// TIA Portal project "Cuptor" (V15.1)

(* hardware
DEVICE "S71500/ET200MP station_1"  S7-1500 station
   slot 0: "Rail_0"  Rack  6ES7 590-1***0-0AA0
   slot 1: "PLC_1"  CPU 1513-1 PN  6ES7 513-1AL02-0AB0  V2.6
      slot 3: "CPU display_1"  6ES7591-1AA00-0AA0
DEVICE "HMI_1"  KTP900 Basic PN
   slot 0: "HMI_1"  KTP900 Basic PN  6AV2 123-2JB03-0AX0  15.1.0.0
   slot 1: "HMI_RT_1"  KTP900 Basic PN  6AV2 123-2JB03-0AX0  15.1.0.0
   slot 5: "HMI_1.IE_CP_1"  PROFINET Interface  15.0.1.0
      slot 1: "PROFINET Interface_1"  PROFINET Interface
         slot 1: "Port_1"  Port
*)

// ===== PLC "PLC_1"  CPU 1513-1 PN =====

VAR_GLOBAL   // PLC tag table "Default tag table"
   "Clock_Byte" AT %MB0 : Byte;
   "Clock_10Hz" AT %M0.0 : Bool;
   "Clock_5Hz" AT %M0.1 : Bool;
   "Clock_2.5Hz" AT %M0.2 : Bool;
   "Clock_2Hz" AT %M0.3 : Bool;
   "Clock_1.25Hz" AT %M0.4 : Bool;
   "Clock_1Hz" AT %M0.5 : Bool;
   "Clock_0.625Hz" AT %M0.6 : Bool;
   "Clock_0.5Hz" AT %M0.7 : Bool;
END_VAR

DATA_BLOCK "Avarii"   // DB1
{ S7_Optimized_Access := 'TRUE' }
VERSION : 0.1
   VAR
      esd : Bool;
      esd_btn : Bool;
      reset_esd_btn : Bool;
      avarie_usa : Bool;
      avarie_trapa : Bool;
      avarie_arzator : Bool;
      avarie_ventilator : Bool;
      avarie_generala : Bool;
      reset_avarie_generala_btn : Bool;
      avarie_hmi : Bool;
      "anti-viagra_pt_al7" : Bool;
   END_VAR
BEGIN
END_DATA_BLOCK

DATA_BLOCK "Usa"   // DB2
{ S7_Optimized_Access := 'TRUE' }
VERSION : 0.1
   VAR
      usa_inchisa : Bool;
      btn_usa_deschisa : Bool;
      btn_usa_deschidere_urgenta : Bool;
   END_VAR
BEGIN
END_DATA_BLOCK

DATA_BLOCK "Trapa"   // DB3
{ S7_Optimized_Access := 'TRUE' }
VERSION : 0.1
   VAR
      trapa_inchisa : Bool;
      btn_trapa_deschisa : Bool;
      btn_trapa_deschidere_urgenta : Bool;
   END_VAR
BEGIN
END_DATA_BLOCK

DATA_BLOCK "Arzator"   // DB4
{ S7_Optimized_Access := 'TRUE' }
VERSION : 0.1
   VAR
      btn_pornire : Bool;
      arzator_pornit : Bool;
   END_VAR
BEGIN
END_DATA_BLOCK

DATA_BLOCK "Ventilator"   // DB5
{ S7_Optimized_Access := 'TRUE' }
VERSION : 0.1
   VAR
      btn_pornire : Bool;
      btn_pornire_urgenta : Bool;
      pornire_stea : Bool;
      pornire_triunghi : Bool;
      pornire_ventilator : Bool;
   END_VAR
BEGIN
END_DATA_BLOCK

DATA_BLOCK "Alarme"   // DB6
{ S7_Optimized_Access := 'TRUE' }
VERSION : 0.1
   VAR
      alarm_gather : Word;
      alarm_vect : Array[0..15] of Bool;
   END_VAR
BEGIN
END_DATA_BLOCK

DATA_BLOCK "Permisiuni"   // DB7
{ S7_Optimized_Access := 'TRUE' }
VERSION : 0.1
   VAR
      permisiune_pornire : Bool;
      cuptor_terminat : Bool;
      timp_50 : Time;
      timp_80 : Time;
      auxiliar_alarma_7 : Bool;
   END_VAR
BEGIN
END_DATA_BLOCK

DATA_BLOCK "Simulare"   // DB10
{ S7_Optimized_Access := 'TRUE' }
VERSION : 0.1
   VAR
      temperatura_curenta : Real;
      temperatura_ceruta : Real;
      temperatura_deschidere : Real := 18.0;
      timp_cuptor : Time;
      resetare_cuptor : Bool;
      timp_curent : Time;
      timp_curent_hmi : Time;
      timp_cuptor_ms : Time;
      add_triunghi : Int;
      paritate_triunghi : Int;
      add_stea : Int;
      paritate_stea : Int;
   END_VAR
BEGIN
END_DATA_BLOCK

DATA_BLOCK "Butoane"   // DB11
{ S7_Optimized_Access := 'TRUE' }
VERSION : 0.1
   VAR
      btn_pornire : Bool;
      btn_pauza : Bool;
      btn_continuare : Bool;
      re_test : Bool;
   END_VAR
BEGIN
END_DATA_BLOCK

DATA_BLOCK "Usa_FB_DB"   // DB12
{ S7_Optimized_Access := 'TRUE' }
VERSION : 0.1
// stored: InstanceOfName Usa_FB
"Usa_FB"
BEGIN
END_DATA_BLOCK

DATA_BLOCK "Trapa_FB_DB"   // DB13
{ S7_Optimized_Access := 'TRUE' }
VERSION : 0.1
// stored: InstanceOfName Trapa_FB
"Trapa_FB"
BEGIN
END_DATA_BLOCK

DATA_BLOCK "Ventilator_FB_DB"   // DB14
{ S7_Optimized_Access := 'TRUE' }
VERSION : 0.1
// stored: InstanceOfName Ventilator_FB
"Ventilator_FB"
BEGIN
END_DATA_BLOCK

DATA_BLOCK "Arzator_FB_DB"   // DB16
{ S7_Optimized_Access := 'TRUE' }
VERSION : 0.1
// stored: InstanceOfName Arzator_FB
"Arzator_FB"
BEGIN
END_DATA_BLOCK

DATA_BLOCK "Simulare_FB_DB"   // DB17
{ S7_Optimized_Access := 'TRUE' }
VERSION : 0.1
// stored: InstanceOfName Simulare_FB
"Simulare_FB"
BEGIN
END_DATA_BLOCK

DATA_BLOCK "Hysteresis_DB_1"   // DB18
{ S7_Optimized_Access := 'TRUE' }
VERSION : 0.1
// stored: InstanceOfName Hysteresis
"Hysteresis"
BEGIN
END_DATA_BLOCK

DATA_BLOCK "Variabile_HMI"   // DB19
{ S7_Optimized_Access := 'TRUE' }
VERSION : 0.1
   VAR
      re_stea : Bool;
      re_triunghi : Bool;
      stea_1 : Bool;
      triunghi_1 : Bool;
      triunghi_2 : Bool;
      stea_2 : Bool;
   END_VAR
BEGIN
END_DATA_BLOCK

// folder: System blocks/Program resources

DATA_BLOCK "Reset_esd"   // DB8
{ S7_Optimized_Access := 'TRUE' }
AUTHOR : Simatic
FAMILY : IEC
NAME : IEC_TMR
VERSION : 1.0
// stored: InstanceOfName IEC_TIMER
"IEC_TIMER"
BEGIN
END_DATA_BLOCK

DATA_BLOCK "Reset_avarie_generala"   // DB9
{ S7_Optimized_Access := 'TRUE' }
AUTHOR : Simatic
FAMILY : IEC
NAME : IEC_TMR
VERSION : 1.0
// stored: InstanceOfName IEC_TIMER
"IEC_TIMER"
BEGIN
END_DATA_BLOCK

DATA_BLOCK "restart_btn_pornire"   // DB15
{ S7_Optimized_Access := 'TRUE' }
AUTHOR : Simatic
FAMILY : IEC
NAME : IEC_TMR
VERSION : 1.0
// stored: InstanceOfName IEC_TIMER
"IEC_TIMER"
BEGIN
END_DATA_BLOCK

// folder: (top level)

FUNCTION_BLOCK "Usa_FB"   // FB1, LAD
{ S7_Optimized_Access := 'TRUE' }
VERSION : 0.1
   VAR_INPUT
      esd : Bool;
      avarie : Bool;
      btn_deschidere_urgenta : Bool;
      temperatura_curenta : Real;
      temperatura_deschidere : Real;
   END_VAR
   VAR_OUTPUT
      usa_inchisa : Bool;
      alarma : Bool;
   END_VAR
   VAR_IN_OUT
      btn_deschidere : Bool;
   END_VAR
   VAR
      timer_reset_alarma : TON_TIME;
   END_VAR
BEGIN

REGION Network 1: Deschide usa(normal sau extrem)
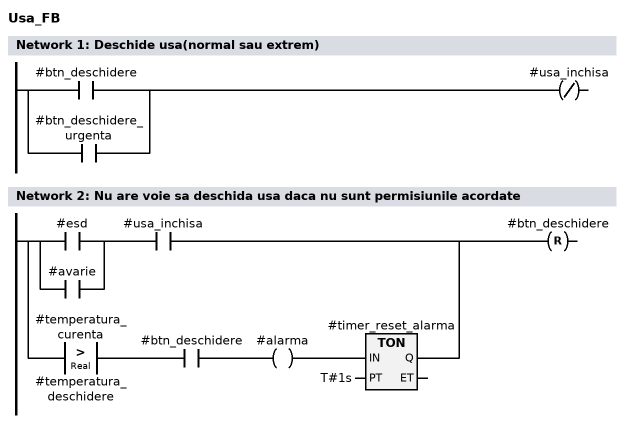
   RUNG wire#powerrail
      Contact( #btn_deschidere )
      wire#w1
      I_Coil( #usa_inchisa )
   END_RUNG
   RUNG wire#powerrail
      Contact( #btn_deschidere_urgenta )
   END_RUNG wire#w1
   // the same network as SCL:
   #usa_inchisa := NOT (#btn_deschidere OR #btn_deschidere_urgenta);
END_REGION

REGION Network 2: Nu are voie sa deschida usa daca nu sunt permisiunile acordate
   #alarma := (#temperatura_curenta > #temperatura_deschidere) AND #btn_deschidere;
   #timer_reset_alarma(IN := #alarma, PT := T#1s);   // TON
   IF ((#esd OR #avarie) AND #usa_inchisa) OR #timer_reset_alarma.Q THEN #btn_deschidere := FALSE; END_IF;
END_REGION
END_FUNCTION_BLOCK

FUNCTION_BLOCK "Trapa_FB"   // FB2, LAD
{ S7_Optimized_Access := 'TRUE' }
VERSION : 0.1
   VAR_INPUT
      esd : Bool;
      avarie : Bool;
      btn_deschidere_urgenta : Bool;
      cuptor_terminat : Bool;
      temperatura_curenta : Real;
      temperatura_inchidere_trapa : Real;
   END_VAR
   VAR_OUTPUT
      trapa_inchisa : Bool;
   END_VAR
   VAR_IN_OUT
      btn_deschidere : Bool;
   END_VAR
BEGIN

REGION Network 1: Deschide trapa(normla si urgenta)
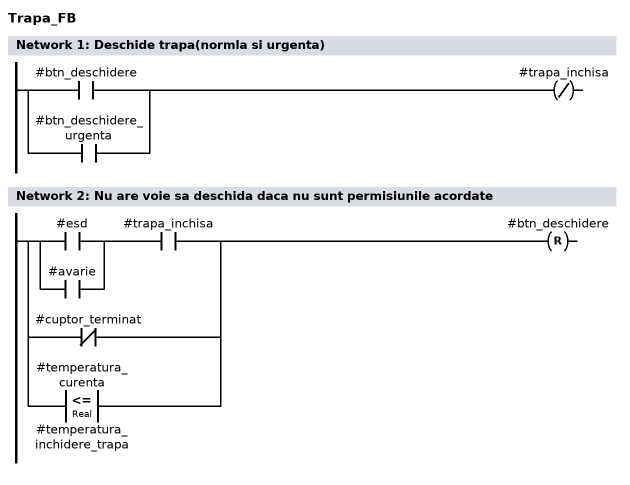
   RUNG wire#powerrail
      Contact( #btn_deschidere )
      wire#w1
      I_Coil( #trapa_inchisa )
   END_RUNG
   RUNG wire#powerrail
      Contact( #btn_deschidere_urgenta )
   END_RUNG wire#w1
   // the same network as SCL:
   #trapa_inchisa := NOT (#btn_deschidere OR #btn_deschidere_urgenta);
END_REGION

REGION Network 2: Nu are voie sa deschida daca nu sunt permisiunile acordate
   RUNG wire#powerrail
      Contact( #esd )
      wire#w1
      Contact( #trapa_inchisa )
      wire#w2
      R_Coil( #btn_deschidere )
   END_RUNG
   RUNG wire#powerrail
      Contact( #avarie )
   END_RUNG wire#w1
   RUNG wire#powerrail
      I_Contact( #cuptor_terminat )
   END_RUNG wire#w2
   RUNG wire#powerrail
      { S7_Templates := "SrcType := Real" } LE_Contact(in1 := #temperatura_curenta, in2 := #temperatura_inchidere_trapa)
   END_RUNG wire#w2
   // the same network as SCL:
   IF ((#esd OR #avarie) AND #trapa_inchisa) OR NOT #cuptor_terminat OR (#temperatura_curenta <= #temperatura_inchidere_trapa) THEN
       #btn_deschidere := FALSE;
   END_IF;
END_REGION
END_FUNCTION_BLOCK

FUNCTION_BLOCK "Arzator_FB"   // FB3, LAD
{ S7_Optimized_Access := 'TRUE' }
VERSION : 0.1
   VAR_INPUT
      esd : Bool;
      avarie : Bool;
      temperatura_curenta : Real;
      temperatura_dorita : Real;
   END_VAR
   VAR_OUTPUT
      pornire_arzator : Bool;
   END_VAR
   VAR_IN_OUT
      btn_pornire : Bool;
   END_VAR
BEGIN

REGION Network 1: Porneste valva
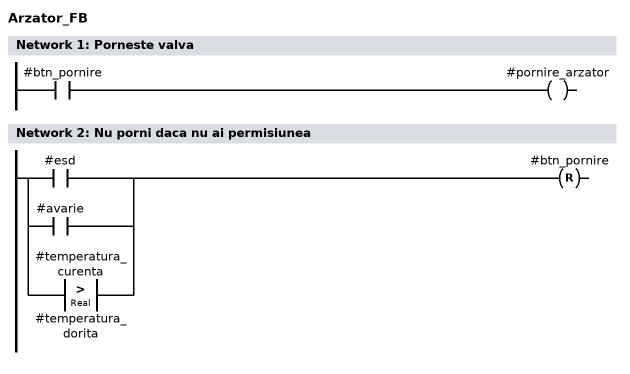
   RUNG wire#powerrail
      Contact( #btn_pornire )
      Coil( #pornire_arzator )
   END_RUNG
   // the same network as SCL:
   #pornire_arzator := #btn_pornire;
END_REGION

REGION Network 2: Nu porni daca nu ai permisiunea
   RUNG wire#powerrail
      Contact( #esd )
      wire#w1
      R_Coil( #btn_pornire )
   END_RUNG
   RUNG wire#powerrail
      Contact( #avarie )
   END_RUNG wire#w1
   RUNG wire#powerrail
      { S7_Templates := "SrcType := Real" } GT_Contact(in1 := #temperatura_curenta, in2 := #temperatura_dorita)
   END_RUNG wire#w1
   // the same network as SCL:
   IF #esd OR #avarie OR (#temperatura_curenta > #temperatura_dorita) THEN #btn_pornire := FALSE; END_IF;
END_REGION
END_FUNCTION_BLOCK

FUNCTION_BLOCK "Ventilator_FB"   // FB4, LAD
{ S7_Optimized_Access := 'TRUE' }
VERSION : 0.1
   VAR_INPUT
      esd : Bool;
      avarie : Bool;
      cuptor_terminat : Bool;
      btn_pornire_urgenta : Bool;
      temperatura_curenta : Real;
      temperatura_inchidere_ventilator : Real;
   END_VAR
   VAR_OUTPUT
      pornire_ventilator_stea : Bool;
      pornire_ventilator_triunghi : Bool;
      ventilator_pornit : Bool;
   END_VAR
   VAR_IN_OUT
      btn_pornire : Bool;
   END_VAR
   VAR
      timer_stea : TON_TIME;
   END_VAR
BEGIN

REGION Network 1: Porneste ventilatorul(normal si urgenta)
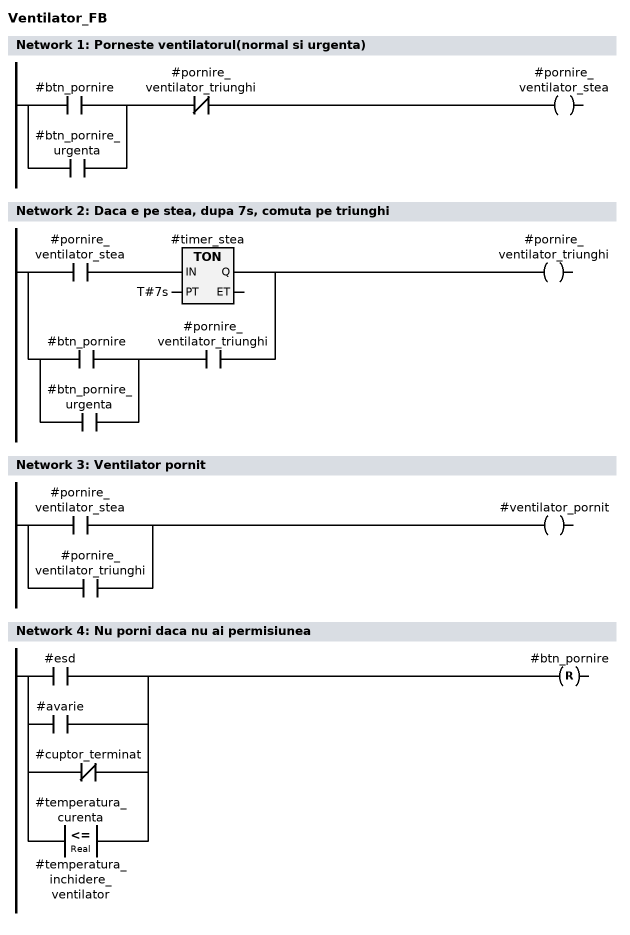
   RUNG wire#powerrail
      Contact( #btn_pornire )
      wire#w1
      I_Contact( #pornire_ventilator_triunghi )
      Coil( #pornire_ventilator_stea )
   END_RUNG
   RUNG wire#powerrail
      Contact( #btn_pornire_urgenta )
   END_RUNG wire#w1
   // the same network as SCL:
   #pornire_ventilator_stea := (#btn_pornire OR #btn_pornire_urgenta) AND NOT #pornire_ventilator_triunghi;
END_REGION

REGION Network 2: Daca e pe stea, dupa 7s, comuta pe triunghi
   #timer_stea(IN := #pornire_ventilator_stea, PT := T#7s);   // TON
   #pornire_ventilator_triunghi := #timer_stea.Q OR ((#btn_pornire OR #btn_pornire_urgenta) AND #pornire_ventilator_triunghi);
END_REGION

REGION Network 3: Ventilator pornit
   RUNG wire#powerrail
      Contact( #pornire_ventilator_stea )
      wire#w1
      Coil( #ventilator_pornit )
   END_RUNG
   RUNG wire#powerrail
      Contact( #pornire_ventilator_triunghi )
   END_RUNG wire#w1
   // the same network as SCL:
   #ventilator_pornit := #pornire_ventilator_stea OR #pornire_ventilator_triunghi;
END_REGION

REGION Network 4: Nu porni daca nu ai permisiunea
   RUNG wire#powerrail
      Contact( #esd )
      wire#w1
      R_Coil( #btn_pornire )
   END_RUNG
   RUNG wire#powerrail
      Contact( #avarie )
   END_RUNG wire#w1
   RUNG wire#powerrail
      I_Contact( #cuptor_terminat )
   END_RUNG wire#w1
   RUNG wire#powerrail
      { S7_Templates := "SrcType := Real" } LE_Contact(in1 := #temperatura_curenta, in2 := #temperatura_inchidere_ventilator)
   END_RUNG wire#w1
   // the same network as SCL:
   IF #esd OR #avarie OR NOT #cuptor_terminat OR (#temperatura_curenta <= #temperatura_inchidere_ventilator) THEN
       #btn_pornire := FALSE;
   END_IF;
END_REGION
END_FUNCTION_BLOCK

FUNCTION_BLOCK "Simulare_FB"   // FB5, LAD
{ S7_Optimized_Access := 'TRUE' }
VERSION : 0.1
   VAR_INPUT
      esd : Bool;
      avarie : Bool;
      temp_dorita : Real;
      temp_mediu : Real := 0.0;
      timp_cuptor : Time;
      trapa : Bool;
      ventilator : Bool;
      ventilator_stea : Bool;
      ventilator_triunghi : Bool;
   END_VAR
   VAR_OUTPUT
      timp_curent : Time;
      btn_trapa : Bool;
      btn_ventilator : Bool;
      terminat : Bool;
      alarma : Bool;
   END_VAR
   VAR_IN_OUT
      resetare_cuptor : Bool;
      temp_curenta : Real;
      pornire_arzator : Bool;
      conditie_pornire : Bool;
   END_VAR
   VAR
      timp_curent_secunde : Time;
      timer_cuptor : TON_TIME;
      re1 : Bool;
      re2 : Bool;
      timp_terminat : Bool;
      temp_in_limite : Bool;
      timer_reset_btn_resetare_cuptor : TON_TIME;
   END_VAR
   VAR_TEMP   // added for the SCL form of the ladder/FBD networks
      _w1 : Bool;
      _w2 : Bool;
      _w3 : Bool;
   END_VAR
BEGIN

REGION Network 1: Daca are permisiunea, da drumul la valva
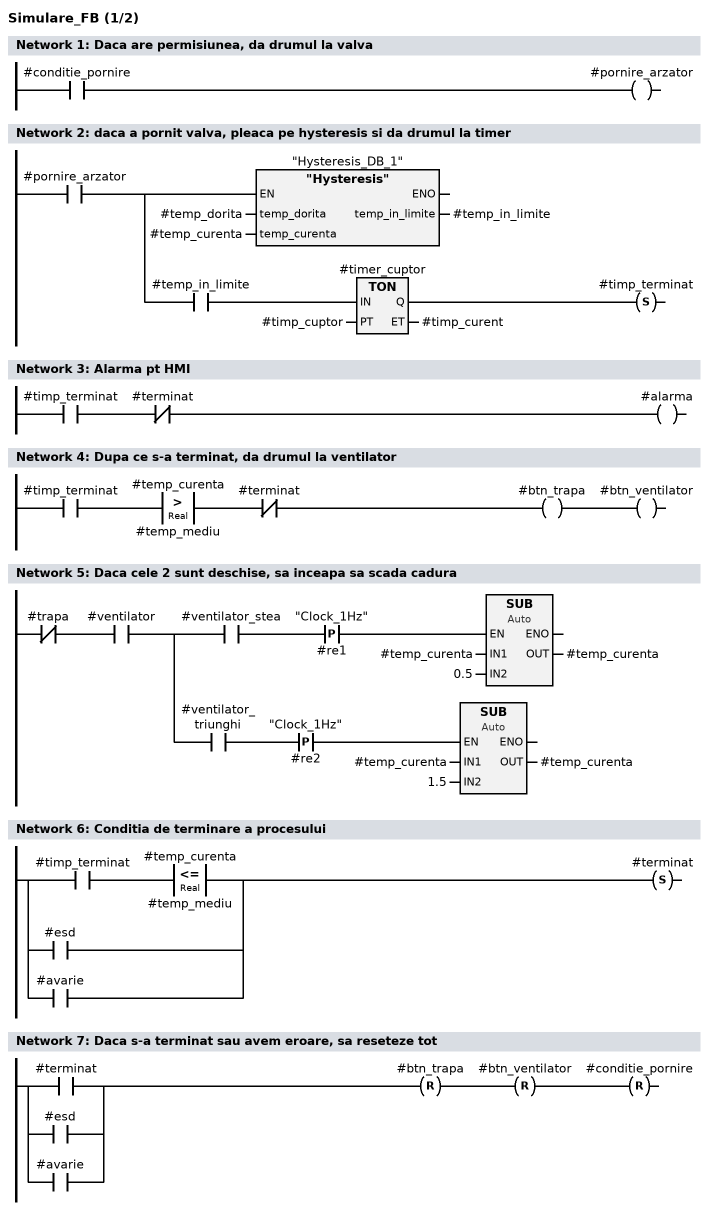
   RUNG wire#powerrail
      Contact( #conditie_pornire )
      Coil( #pornire_arzator )
   END_RUNG
   // the same network as SCL:
   #pornire_arzator := #conditie_pornire;
END_REGION

REGION Network 2: daca a pornit valva, pleaca pe hysteresis si da drumul la timer
   IF #pornire_arzator THEN
       "Hysteresis_DB_1"(temp_dorita := #temp_dorita,   // "Hysteresis"
                         temp_curenta := #temp_curenta,
                         temp_in_limite => #temp_in_limite);
   END_IF;
   #timer_cuptor(IN := #pornire_arzator AND #temp_in_limite, PT := #timp_cuptor, ET => #timp_curent);   // TON
   IF #timer_cuptor.Q THEN #timp_terminat := TRUE; END_IF;
END_REGION

REGION Network 3: Alarma pt HMI
   RUNG wire#powerrail
      Contact( #timp_terminat )
      I_Contact( #terminat )
      Coil( #alarma )
   END_RUNG
   // the same network as SCL:
   #alarma := #timp_terminat AND NOT #terminat;
END_REGION

REGION Network 4: Dupa ce s-a terminat, da drumul la ventilator
   RUNG wire#powerrail
      Contact( #timp_terminat )
      { S7_Templates := "SrcType := Real" } GT_Contact(in1 := #temp_curenta, in2 := #temp_mediu)
      I_Contact( #terminat )
      Coil( #btn_trapa )
      Coil( #btn_ventilator )
   END_RUNG
   // the same network as SCL:
   #btn_trapa := #timp_terminat AND (#temp_curenta > #temp_mediu) AND NOT #terminat;
   #btn_ventilator := #btn_trapa;
END_REGION

REGION Network 5: Daca cele 2 sunt deschise, sa inceapa sa scada cadura
   RUNG wire#powerrail
      I_Contact( #trapa )
      Contact( #ventilator )
      wire#w1
      Contact( #ventilator_stea )
      P_Contact(operand := "Clock_1Hz", bit := #re1)
      Sub(in1 := #temp_curenta, in2 := 0.5, out => #temp_curenta)
   END_RUNG
   RUNG wire#w1
      Contact( #ventilator_triunghi )
      P_Contact(operand := "Clock_1Hz", bit := #re2)
      Sub(in1 := #temp_curenta, in2 := 1.5, out => #temp_curenta)
   END_RUNG
   // the same network as SCL:
   #_w1 := NOT #trapa AND #ventilator;
   #_w2 := #_w1 AND #ventilator_stea AND "Clock_1Hz" AND NOT #re1;   // rising edge of "Clock_1Hz"
   #re1 := "Clock_1Hz";
   IF #_w2 THEN #temp_curenta := #temp_curenta - 0.5; END_IF;
   #_w3 := #_w1 AND #ventilator_triunghi AND "Clock_1Hz" AND NOT #re2;   // rising edge of "Clock_1Hz"
   #re2 := "Clock_1Hz";
   IF #_w3 THEN #temp_curenta := #temp_curenta - 1.5; END_IF;
END_REGION

REGION Network 6: Conditia de terminare a procesului
   RUNG wire#powerrail
      Contact( #timp_terminat )
      { S7_Templates := "SrcType := Real" } LE_Contact(in1 := #temp_curenta, in2 := #temp_mediu)
      wire#w1
      S_Coil( #terminat )
   END_RUNG
   RUNG wire#powerrail
      Contact( #esd )
   END_RUNG wire#w1
   RUNG wire#powerrail
      Contact( #avarie )
   END_RUNG wire#w1
   // the same network as SCL:
   IF (#timp_terminat AND (#temp_curenta <= #temp_mediu)) OR #esd OR #avarie THEN #terminat := TRUE; END_IF;
END_REGION

REGION Network 7: Daca s-a terminat sau avem eroare, sa reseteze tot
   RUNG wire#powerrail
      Contact( #terminat )
      wire#w1
      R_Coil( #btn_trapa )
      R_Coil( #btn_ventilator )
      R_Coil( #conditie_pornire )
   END_RUNG
   RUNG wire#powerrail
      Contact( #esd )
   END_RUNG wire#w1
   RUNG wire#powerrail
      Contact( #avarie )
   END_RUNG wire#w1
   // the same network as SCL:
   IF #terminat OR #esd OR #avarie THEN
       #btn_trapa := FALSE;
       #btn_ventilator := FALSE;
       #conditie_pornire := FALSE;
   END_IF;
END_REGION

REGION Network 8: Resetare cuptor
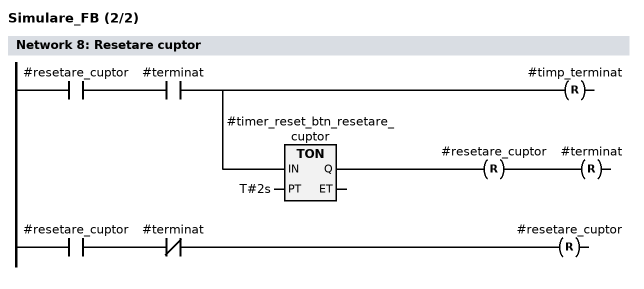
   #_w1 := #resetare_cuptor AND #terminat;
   IF #_w1 THEN #timp_terminat := FALSE; END_IF;
   #timer_reset_btn_resetare_cuptor(IN := #_w1, PT := T#2s);   // TON
   IF #timer_reset_btn_resetare_cuptor.Q THEN
       #resetare_cuptor := FALSE;
       #terminat := FALSE;
   END_IF;
   IF #resetare_cuptor AND NOT #terminat THEN #resetare_cuptor := FALSE; END_IF;
END_REGION
END_FUNCTION_BLOCK

FUNCTION_BLOCK "Hysteresis"   // FB6, LAD
{ S7_Optimized_Access := 'TRUE' }
VERSION : 0.1
   VAR_INPUT
      temp_dorita : Real;
   END_VAR
   VAR_OUTPUT
      temp_in_limite : Bool;
   END_VAR
   VAR_IN_OUT
      temp_curenta : Real;
   END_VAR
   VAR
      crestere_temp : Real := 0.5;
      limita_inferioara : Real;
      limita_superioara : Real;
      differenta_pt_limite : Real := 2.0;
      re1 : Bool;
      re2 : Bool;
      urcare : Bool;
      coborare : Bool;
   END_VAR
   VAR_TEMP   // added for the SCL form of the ladder/FBD networks
      _w1 : Bool;
   END_VAR
BEGIN

REGION Network 1: Calcul pentru limite
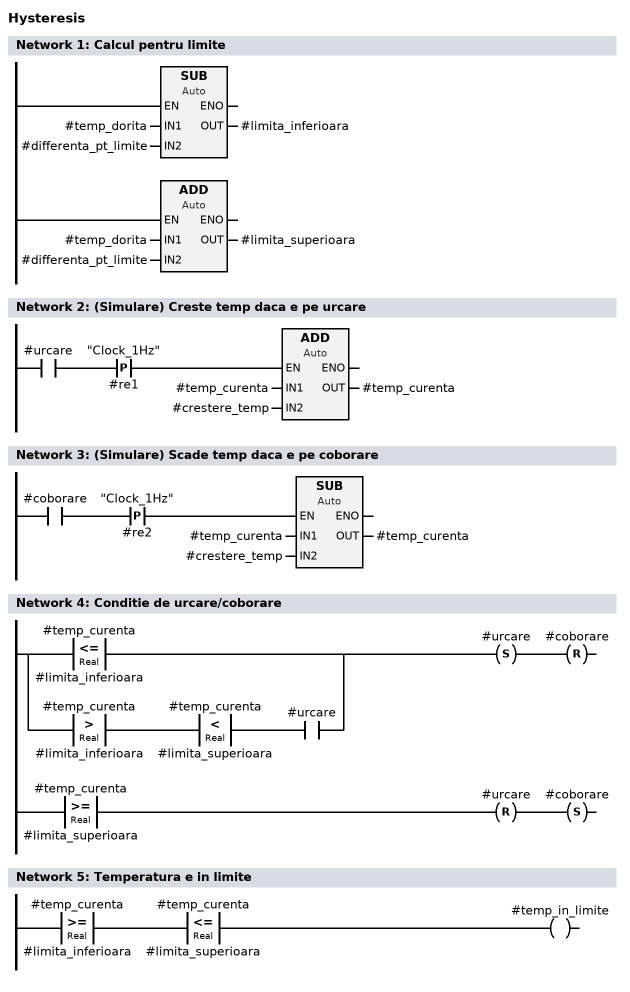
   RUNG wire#powerrail
      Sub(in1 := #temp_dorita, in2 := #differenta_pt_limite, out => #limita_inferioara)
   END_RUNG
   RUNG wire#powerrail
      Add(in1 := #temp_dorita, in2 := #differenta_pt_limite, out => #limita_superioara)
   END_RUNG
   // the same network as SCL:
   #limita_inferioara := #temp_dorita - #differenta_pt_limite;
   #limita_superioara := #temp_dorita + #differenta_pt_limite;
END_REGION

REGION Network 2: (Simulare) Creste temp daca e pe urcare
   RUNG wire#powerrail
      Contact( #urcare )
      P_Contact(operand := "Clock_1Hz", bit := #re1)
      Add(in1 := #temp_curenta, in2 := #crestere_temp, out => #temp_curenta)
   END_RUNG
   // the same network as SCL:
   #_w1 := #urcare AND "Clock_1Hz" AND NOT #re1;   // rising edge of "Clock_1Hz"
   #re1 := "Clock_1Hz";
   IF #_w1 THEN #temp_curenta := #temp_curenta + #crestere_temp; END_IF;
END_REGION

REGION Network 3: (Simulare) Scade temp daca e pe coborare
   RUNG wire#powerrail
      Contact( #coborare )
      P_Contact(operand := "Clock_1Hz", bit := #re2)
      Sub(in1 := #temp_curenta, in2 := #crestere_temp, out => #temp_curenta)
   END_RUNG
   // the same network as SCL:
   #_w1 := #coborare AND "Clock_1Hz" AND NOT #re2;   // rising edge of "Clock_1Hz"
   #re2 := "Clock_1Hz";
   IF #_w1 THEN #temp_curenta := #temp_curenta - #crestere_temp; END_IF;
END_REGION

REGION Network 4: Conditie de urcare/coborare
   RUNG wire#powerrail
      { S7_Templates := "SrcType := Real" } LE_Contact(in1 := #temp_curenta, in2 := #limita_inferioara)
      wire#w1
      S_Coil( #urcare )
      R_Coil( #coborare )
   END_RUNG
   RUNG wire#powerrail
      { S7_Templates := "SrcType := Real" } GT_Contact(in1 := #temp_curenta, in2 := #limita_inferioara)
      { S7_Templates := "SrcType := Real" } LT_Contact(in1 := #temp_curenta, in2 := #limita_superioara)
      Contact( #urcare )
   END_RUNG wire#w1
   RUNG wire#powerrail
      { S7_Templates := "SrcType := Real" } GE_Contact(in1 := #temp_curenta, in2 := #limita_superioara)
      R_Coil( #urcare )
      S_Coil( #coborare )
   END_RUNG
   // the same network as SCL:
   #_w1 := (#temp_curenta <= #limita_inferioara) OR ((#temp_curenta > #limita_inferioara) AND (#temp_curenta < #limita_superioara) AND #urcare);
   IF #_w1 THEN
       #urcare := TRUE;
       #coborare := FALSE;
   END_IF;
   IF #temp_curenta >= #limita_superioara THEN
       #urcare := FALSE;
       #coborare := TRUE;
   END_IF;
END_REGION

REGION Network 5: Temperatura e in limite
   RUNG wire#powerrail
      { S7_Templates := "SrcType := Real" } GE_Contact(in1 := #temp_curenta, in2 := #limita_inferioara)
      { S7_Templates := "SrcType := Real" } LE_Contact(in1 := #temp_curenta, in2 := #limita_superioara)
      Coil( #temp_in_limite )
   END_RUNG
   // the same network as SCL:
   #temp_in_limite := (#temp_curenta >= #limita_inferioara) AND (#temp_curenta <= #limita_superioara);
END_REGION
END_FUNCTION_BLOCK

ORGANIZATION_BLOCK "Main"   // OB1, LAD, ProgramCycle
TITLE = "Main Program Sweep (Cycle)"
{ S7_Optimized_Access := 'TRUE' }
VERSION : 0.1
   VAR_INPUT
      Initial_Call : Bool;   // Initial call of this OB
      Remanence : Bool;   // =True, if remanent data are available
   END_VAR
   VAR_TEMP   // added for the SCL form of the ladder/FBD networks
      _w1 : Bool;
      _w2 : Bool;
   END_VAR
BEGIN

REGION Network 1: Gather pt alarme
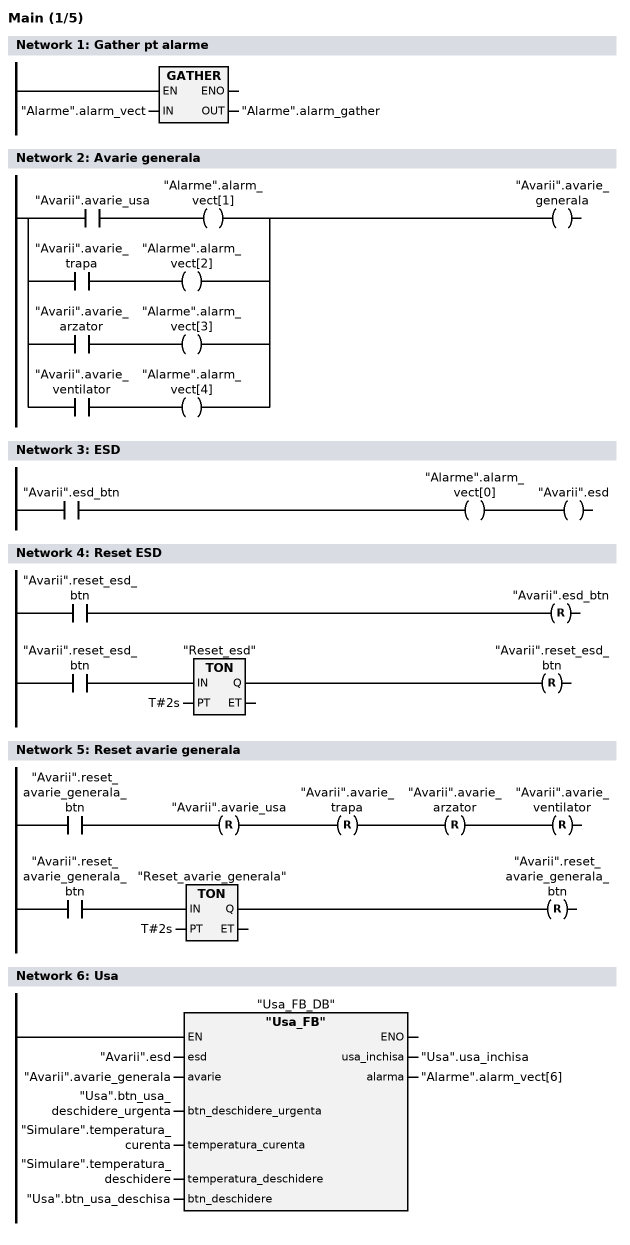
   GATHER(IN := "Alarme".alarm_vect, OUT => "Alarme".alarm_gather);
END_REGION

REGION Network 2: Avarie generala
   RUNG wire#powerrail
      Contact( "Avarii".avarie_usa )
      Coil( "Alarme".alarm_vect[1] )
      wire#w1
      Coil( "Avarii".avarie_generala )
   END_RUNG
   RUNG wire#powerrail
      Contact( "Avarii".avarie_trapa )
      Coil( "Alarme".alarm_vect[2] )
   END_RUNG wire#w1
   RUNG wire#powerrail
      Contact( "Avarii".avarie_arzator )
      Coil( "Alarme".alarm_vect[3] )
   END_RUNG wire#w1
   RUNG wire#powerrail
      Contact( "Avarii".avarie_ventilator )
      Coil( "Alarme".alarm_vect[4] )
   END_RUNG wire#w1
   // the same network as SCL:
   "Alarme".alarm_vect[1] := "Avarii".avarie_usa;
   "Alarme".alarm_vect[2] := "Avarii".avarie_trapa;
   "Alarme".alarm_vect[3] := "Avarii".avarie_arzator;
   "Alarme".alarm_vect[4] := "Avarii".avarie_ventilator;
   "Avarii".avarie_generala := "Avarii".avarie_usa OR "Avarii".avarie_trapa OR "Avarii".avarie_arzator OR "Avarii".avarie_ventilator;
END_REGION

REGION Network 3: ESD
   RUNG wire#powerrail
      Contact( "Avarii".esd_btn )
      Coil( "Alarme".alarm_vect[0] )
      Coil( "Avarii".esd )
   END_RUNG
   // the same network as SCL:
   "Alarme".alarm_vect[0] := "Avarii".esd_btn;
   "Avarii".esd := "Avarii".esd_btn;
END_REGION

REGION Network 4: Reset ESD
   IF "Avarii".reset_esd_btn THEN "Avarii".esd_btn := FALSE; END_IF;
   "Reset_esd".TON(IN := "Avarii".reset_esd_btn, PT := T#2s);
   IF "Reset_esd".Q THEN "Avarii".reset_esd_btn := FALSE; END_IF;
END_REGION

REGION Network 5: Reset avarie generala
   IF "Avarii".reset_avarie_generala_btn THEN
       "Avarii".avarie_usa := FALSE;
       "Avarii".avarie_trapa := FALSE;
       "Avarii".avarie_arzator := FALSE;
       "Avarii".avarie_ventilator := FALSE;
   END_IF;
   "Reset_avarie_generala".TON(IN := "Avarii".reset_avarie_generala_btn, PT := T#2s);
   IF "Reset_avarie_generala".Q THEN "Avarii".reset_avarie_generala_btn := FALSE; END_IF;
END_REGION

REGION Network 6: Usa
   RUNG wire#powerrail
      "Usa_FB_DB"(esd := "Avarii".esd, avarie := "Avarii".avarie_generala, btn_deschidere_urgenta := "Usa".btn_usa_deschidere_urgenta, temperatura_curenta := "Simulare".temperatura_curenta, temperatura_deschidere := "Simulare".temperatura_deschidere, btn_deschidere := "Usa".btn_usa_deschisa, usa_inchisa => "Usa".usa_inchisa, alarma => "Alarme".alarm_vect[6])
   END_RUNG
   // the same network as SCL:
   "Usa_FB_DB"(esd := "Avarii".esd,   // "Usa_FB"
               avarie := "Avarii".avarie_generala,
               btn_deschidere_urgenta := "Usa".btn_usa_deschidere_urgenta,
               temperatura_curenta := "Simulare".temperatura_curenta,
               temperatura_deschidere := "Simulare".temperatura_deschidere,
               btn_deschidere := "Usa".btn_usa_deschisa,
               usa_inchisa => "Usa".usa_inchisa,
               alarma => "Alarme".alarm_vect[6]);
END_REGION

REGION Network 7: Trapa
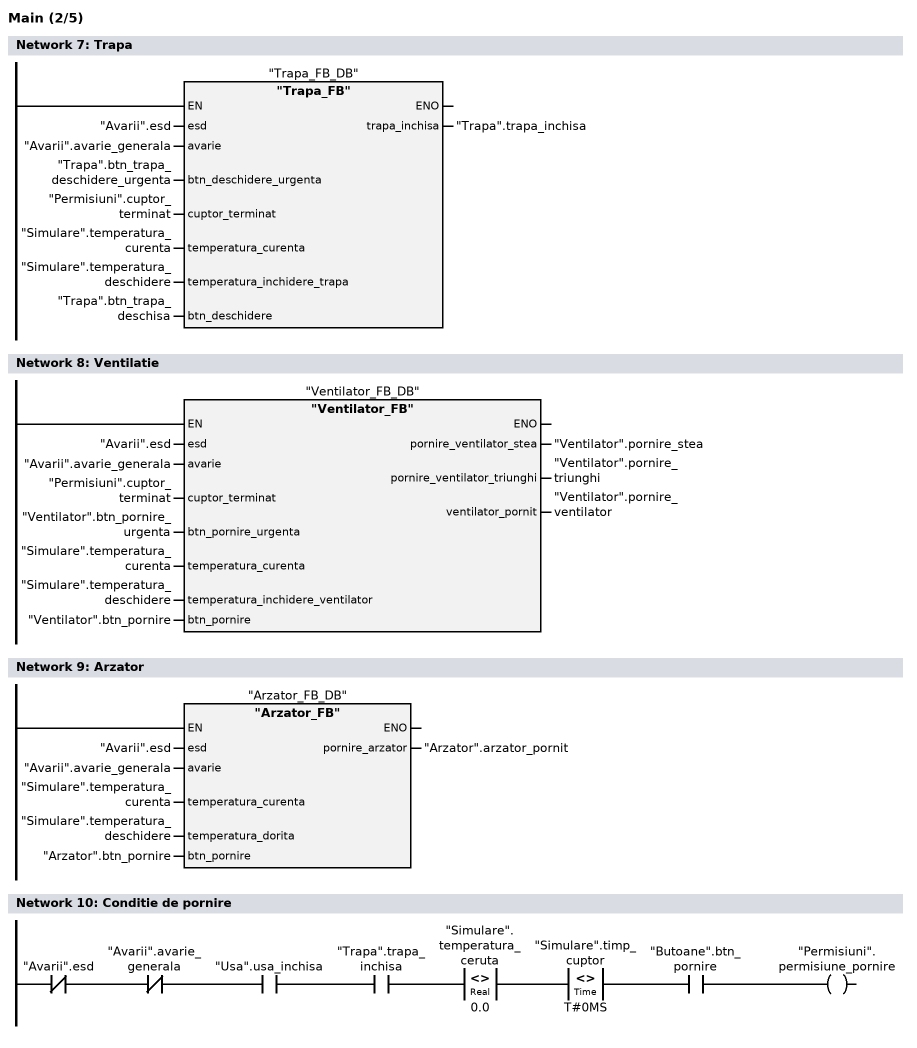
   RUNG wire#powerrail
      "Trapa_FB_DB"(esd := "Avarii".esd, avarie := "Avarii".avarie_generala, btn_deschidere_urgenta := "Trapa".btn_trapa_deschidere_urgenta, cuptor_terminat := "Permisiuni".cuptor_terminat, temperatura_curenta := "Simulare".temperatura_curenta, temperatura_inchidere_trapa := "Simulare".temperatura_deschidere, btn_deschidere := "Trapa".btn_trapa_deschisa, trapa_inchisa => "Trapa".trapa_inchisa)
   END_RUNG
   // the same network as SCL:
   "Trapa_FB_DB"(esd := "Avarii".esd,   // "Trapa_FB"
                 avarie := "Avarii".avarie_generala,
                 btn_deschidere_urgenta := "Trapa".btn_trapa_deschidere_urgenta,
                 cuptor_terminat := "Permisiuni".cuptor_terminat,
                 temperatura_curenta := "Simulare".temperatura_curenta,
                 temperatura_inchidere_trapa := "Simulare".temperatura_deschidere,
                 btn_deschidere := "Trapa".btn_trapa_deschisa,
                 trapa_inchisa => "Trapa".trapa_inchisa);
END_REGION

REGION Network 8: Ventilatie
   RUNG wire#powerrail
      "Ventilator_FB_DB"(esd := "Avarii".esd, avarie := "Avarii".avarie_generala, cuptor_terminat := "Permisiuni".cuptor_terminat, btn_pornire_urgenta := "Ventilator".btn_pornire_urgenta, temperatura_curenta := "Simulare".temperatura_curenta, temperatura_inchidere_ventilator := "Simulare".temperatura_deschidere, btn_pornire := "Ventilator".btn_pornire, pornire_ventilator_stea => "Ventilator".pornire_stea, pornire_ventilator_triunghi => "Ventilator".pornire_triunghi, ventilator_pornit => "Ventilator".pornire_ventilator)
   END_RUNG
   // the same network as SCL:
   "Ventilator_FB_DB"(esd := "Avarii".esd,   // "Ventilator_FB"
                      avarie := "Avarii".avarie_generala,
                      cuptor_terminat := "Permisiuni".cuptor_terminat,
                      btn_pornire_urgenta := "Ventilator".btn_pornire_urgenta,
                      temperatura_curenta := "Simulare".temperatura_curenta,
                      temperatura_inchidere_ventilator := "Simulare".temperatura_deschidere,
                      btn_pornire := "Ventilator".btn_pornire,
                      pornire_ventilator_stea => "Ventilator".pornire_stea,
                      pornire_ventilator_triunghi => "Ventilator".pornire_triunghi,
                      ventilator_pornit => "Ventilator".pornire_ventilator);
END_REGION

REGION Network 9: Arzator
   RUNG wire#powerrail
      "Arzator_FB_DB"(esd := "Avarii".esd, avarie := "Avarii".avarie_generala, temperatura_curenta := "Simulare".temperatura_curenta, temperatura_dorita := "Simulare".temperatura_deschidere, btn_pornire := "Arzator".btn_pornire, pornire_arzator => "Arzator".arzator_pornit)
   END_RUNG
   // the same network as SCL:
   "Arzator_FB_DB"(esd := "Avarii".esd,   // "Arzator_FB"
                   avarie := "Avarii".avarie_generala,
                   temperatura_curenta := "Simulare".temperatura_curenta,
                   temperatura_dorita := "Simulare".temperatura_deschidere,
                   btn_pornire := "Arzator".btn_pornire,
                   pornire_arzator => "Arzator".arzator_pornit);
END_REGION

REGION Network 10: Conditie de pornire
   RUNG wire#powerrail
      I_Contact( "Avarii".esd )
      I_Contact( "Avarii".avarie_generala )
      Contact( "Usa".usa_inchisa )
      Contact( "Trapa".trapa_inchisa )
      { S7_Templates := "SrcType := Real" } NE_Contact(in1 := "Simulare".temperatura_ceruta, in2 := 0.0)
      { S7_Templates := "SrcType := Time" } NE_Contact(in1 := "Simulare".timp_cuptor, in2 := T#0MS)
      Contact( "Butoane".btn_pornire )
      Coil( "Permisiuni".permisiune_pornire )
   END_RUNG
   // the same network as SCL:
   "Permisiuni".permisiune_pornire := NOT "Avarii".esd AND NOT "Avarii".avarie_generala AND "Usa".usa_inchisa AND "Trapa".trapa_inchisa AND ("Simulare".temperatura_ceruta <> 0.0) AND ("Simulare".timp_cuptor <> T#0MS) AND "Butoane".btn_pornire;
END_REGION

REGION Network 11: Alarme
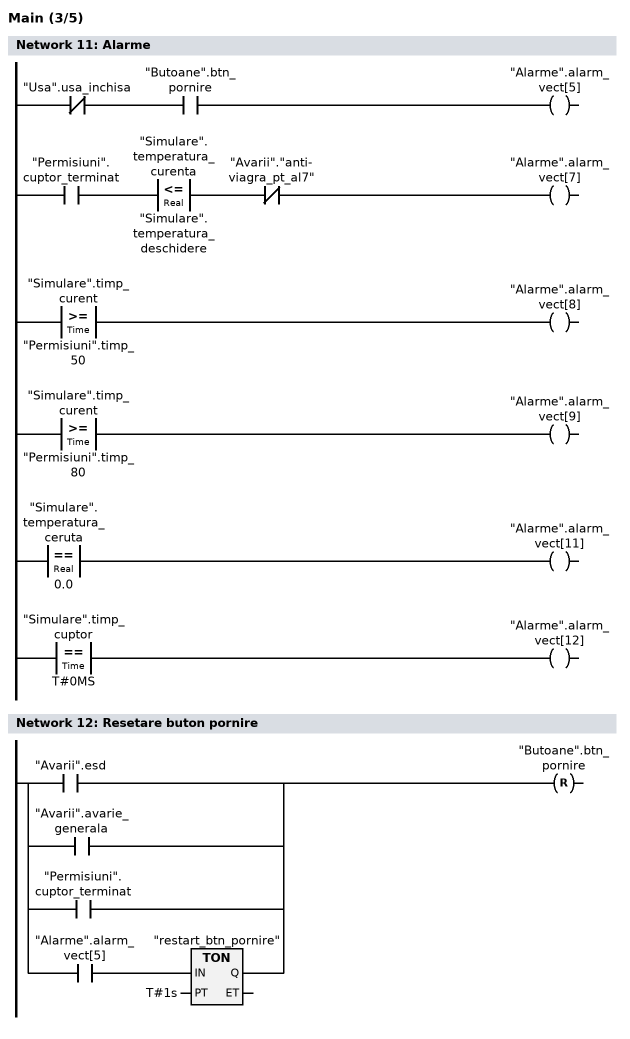
   RUNG wire#powerrail
      I_Contact( "Usa".usa_inchisa )
      Contact( "Butoane".btn_pornire )
      Coil( "Alarme".alarm_vect[5] )
   END_RUNG
   RUNG wire#powerrail
      Contact( "Permisiuni".cuptor_terminat )
      { S7_Templates := "SrcType := Real" } LE_Contact(in1 := "Simulare".temperatura_curenta, in2 := "Simulare".temperatura_deschidere)
      I_Contact( "Avarii"."anti-viagra_pt_al7" )
      Coil( "Alarme".alarm_vect[7] )
   END_RUNG
   RUNG wire#powerrail
      { S7_Templates := "SrcType := Time" } GE_Contact(in1 := "Simulare".timp_curent, in2 := "Permisiuni".timp_50)
      Coil( "Alarme".alarm_vect[8] )
   END_RUNG
   RUNG wire#powerrail
      { S7_Templates := "SrcType := Time" } GE_Contact(in1 := "Simulare".timp_curent, in2 := "Permisiuni".timp_80)
      Coil( "Alarme".alarm_vect[9] )
   END_RUNG
   RUNG wire#powerrail
      { S7_Templates := "SrcType := Real" } EQ_Contact(in1 := "Simulare".temperatura_ceruta, in2 := 0.0)
      Coil( "Alarme".alarm_vect[11] )
   END_RUNG
   RUNG wire#powerrail
      { S7_Templates := "SrcType := Time" } EQ_Contact(in1 := "Simulare".timp_cuptor, in2 := T#0MS)
      Coil( "Alarme".alarm_vect[12] )
   END_RUNG
   // the same network as SCL:
   "Alarme".alarm_vect[5] := NOT "Usa".usa_inchisa AND "Butoane".btn_pornire;
   "Alarme".alarm_vect[7] := "Permisiuni".cuptor_terminat AND ("Simulare".temperatura_curenta <= "Simulare".temperatura_deschidere) AND NOT "Avarii"."anti-viagra_pt_al7";
   "Alarme".alarm_vect[8] := "Simulare".timp_curent >= "Permisiuni".timp_50;
   "Alarme".alarm_vect[9] := "Simulare".timp_curent >= "Permisiuni".timp_80;
   "Alarme".alarm_vect[11] := "Simulare".temperatura_ceruta = 0.0;
   "Alarme".alarm_vect[12] := "Simulare".timp_cuptor = T#0MS;
END_REGION

REGION Network 12: Resetare buton pornire
   "restart_btn_pornire".TON(IN := "Alarme".alarm_vect[5], PT := T#1s);
   IF "Avarii".esd OR "Avarii".avarie_generala OR "Permisiuni".cuptor_terminat OR "restart_btn_pornire".Q THEN
       "Butoane".btn_pornire := FALSE;
   END_IF;
END_REGION

REGION Network 13: Simulare
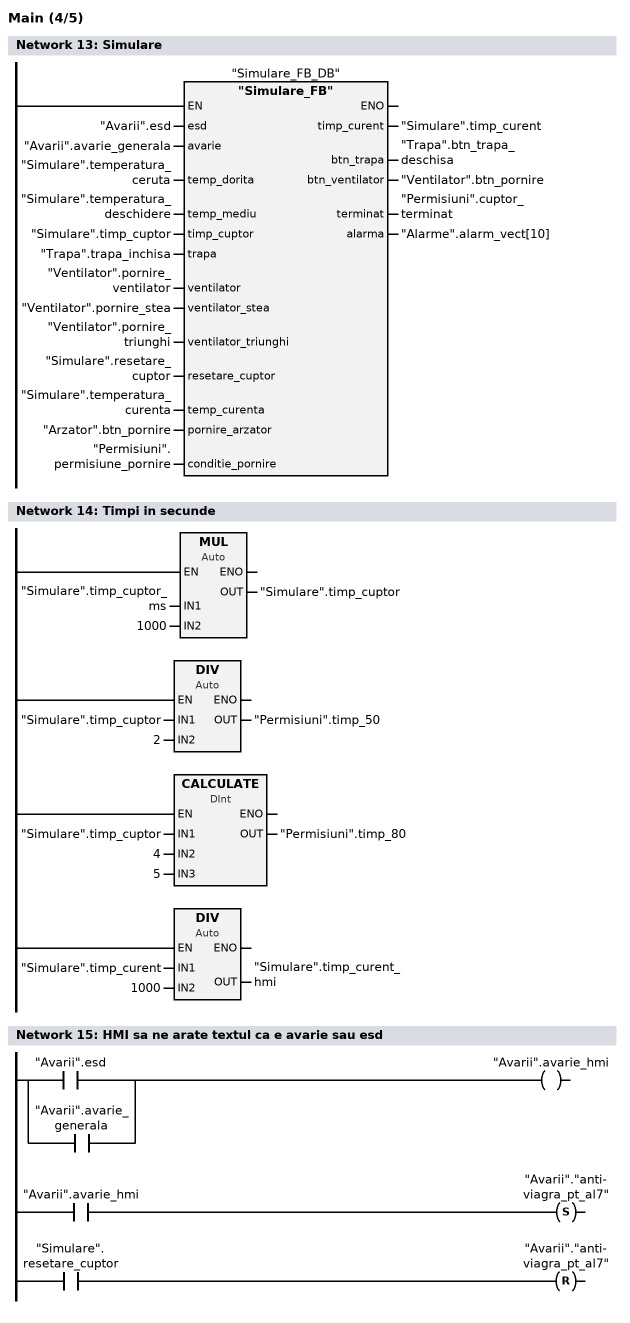
   RUNG wire#powerrail
      "Simulare_FB_DB"(esd := "Avarii".esd, avarie := "Avarii".avarie_generala, temp_dorita := "Simulare".temperatura_ceruta, temp_mediu := "Simulare".temperatura_deschidere, timp_cuptor := "Simulare".timp_cuptor, trapa := "Trapa".trapa_inchisa, ventilator := "Ventilator".pornire_ventilator, ventilator_stea := "Ventilator".pornire_stea, ventilator_triunghi := "Ventilator".pornire_triunghi, resetare_cuptor := "Simulare".resetare_cuptor, temp_curenta := "Simulare".temperatura_curenta, pornire_arzator := "Arzator".btn_pornire, conditie_pornire := "Permisiuni".permisiune_pornire, timp_curent => "Simulare".timp_curent, btn_trapa => "Trapa".btn_trapa_deschisa, btn_ventilator => "Ventilator".btn_pornire, terminat => "Permisiuni".cuptor_terminat, alarma => "Alarme".alarm_vect[10])
   END_RUNG
   // the same network as SCL:
   "Simulare_FB_DB"(esd := "Avarii".esd,   // "Simulare_FB"
                    avarie := "Avarii".avarie_generala,
                    temp_dorita := "Simulare".temperatura_ceruta,
                    temp_mediu := "Simulare".temperatura_deschidere,
                    timp_cuptor := "Simulare".timp_cuptor,
                    trapa := "Trapa".trapa_inchisa,
                    ventilator := "Ventilator".pornire_ventilator,
                    ventilator_stea := "Ventilator".pornire_stea,
                    ventilator_triunghi := "Ventilator".pornire_triunghi,
                    resetare_cuptor := "Simulare".resetare_cuptor,
                    temp_curenta := "Simulare".temperatura_curenta,
                    pornire_arzator := "Arzator".btn_pornire,
                    conditie_pornire := "Permisiuni".permisiune_pornire,
                    timp_curent => "Simulare".timp_curent,
                    btn_trapa => "Trapa".btn_trapa_deschisa,
                    btn_ventilator => "Ventilator".btn_pornire,
                    terminat => "Permisiuni".cuptor_terminat,
                    alarma => "Alarme".alarm_vect[10]);
END_REGION

REGION Network 14: Timpi in secunde
   RUNG wire#powerrail
      Mul(in1 := "Simulare".timp_cuptor_ms, in2 := 1000, out => "Simulare".timp_cuptor)
   END_RUNG
   RUNG wire#powerrail
      Div(in1 := "Simulare".timp_cuptor, in2 := 2, out => "Permisiuni".timp_50)
   END_RUNG
   RUNG wire#powerrail
      { S7_Templates := "SrcType := DInt"; S7_Expression := "IN1* IN2 / IN3" } Calculate(in1 := "Simulare".timp_cuptor, in2 := 4, in3 := 5, out => "Permisiuni".timp_80)
   END_RUNG
   RUNG wire#powerrail
      Div(in1 := "Simulare".timp_curent, in2 := 1000, out => "Simulare".timp_curent_hmi)
   END_RUNG
   // the same network as SCL:
   "Simulare".timp_cuptor := "Simulare".timp_cuptor_ms * 1000;
   "Permisiuni".timp_50 := "Simulare".timp_cuptor / 2;
   "Permisiuni".timp_80 := "Simulare".timp_cuptor* 4 / 5;
   "Simulare".timp_curent_hmi := "Simulare".timp_curent / 1000;
END_REGION

REGION Network 15: HMI sa ne arate textul ca e avarie sau esd
   RUNG wire#powerrail
      Contact( "Avarii".esd )
      wire#w1
      Coil( "Avarii".avarie_hmi )
   END_RUNG
   RUNG wire#powerrail
      Contact( "Avarii".avarie_generala )
   END_RUNG wire#w1
   RUNG wire#powerrail
      Contact( "Avarii".avarie_hmi )
      S_Coil( "Avarii"."anti-viagra_pt_al7" )
   END_RUNG
   RUNG wire#powerrail
      Contact( "Simulare".resetare_cuptor )
      R_Coil( "Avarii"."anti-viagra_pt_al7" )
   END_RUNG
   // the same network as SCL:
   "Avarii".avarie_hmi := "Avarii".esd OR "Avarii".avarie_generala;
   IF "Avarii".avarie_hmi THEN "Avarii"."anti-viagra_pt_al7" := TRUE; END_IF;
   IF "Simulare".resetare_cuptor THEN "Avarii"."anti-viagra_pt_al7" := FALSE; END_IF;
END_REGION

REGION Network 16: HMI ventilator stea
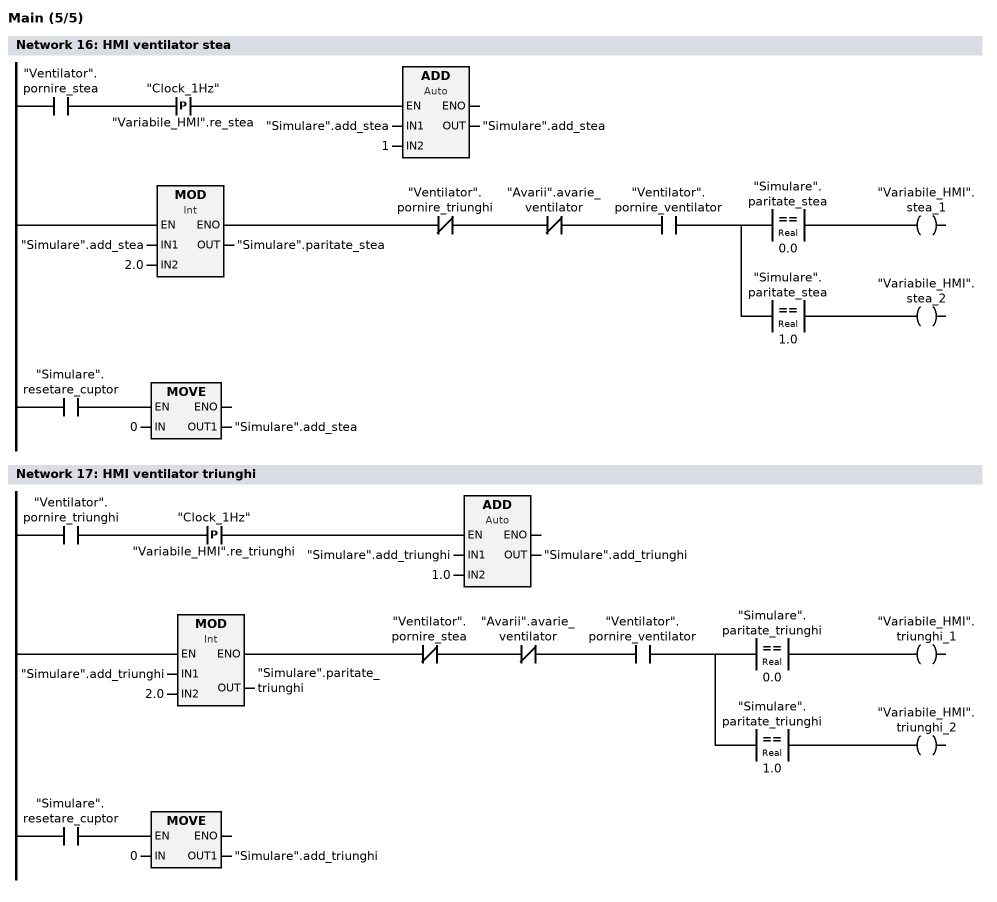
   RUNG wire#powerrail
      Contact( "Ventilator".pornire_stea )
      P_Contact(operand := "Clock_1Hz", bit := "Variabile_HMI".re_stea)
      Add(in1 := "Simulare".add_stea, in2 := 1, out => "Simulare".add_stea)
   END_RUNG
   RUNG wire#powerrail
      { S7_Templates := "SrcType := Int" } Mod(in1 := "Simulare".add_stea, in2 := 2.0, out => "Simulare".paritate_stea)
      I_Contact( "Ventilator".pornire_triunghi )
      I_Contact( "Avarii".avarie_ventilator )
      Contact( "Ventilator".pornire_ventilator )
      wire#w1
      { S7_Templates := "SrcType := Real" } EQ_Contact(in1 := "Simulare".paritate_stea, in2 := 0.0)
      Coil( "Variabile_HMI".stea_1 )
   END_RUNG
   RUNG wire#w1
      { S7_Templates := "SrcType := Real" } EQ_Contact(in1 := "Simulare".paritate_stea, in2 := 1.0)
      Coil( "Variabile_HMI".stea_2 )
   END_RUNG
   RUNG wire#powerrail
      Contact( "Simulare".resetare_cuptor )
      Move(in := 0, out1 => "Simulare".add_stea)
   END_RUNG
   // the same network as SCL:
   #_w1 := "Ventilator".pornire_stea AND "Clock_1Hz" AND NOT "Variabile_HMI".re_stea;   // rising edge of "Clock_1Hz"
   "Variabile_HMI".re_stea := "Clock_1Hz";
   IF #_w1 THEN "Simulare".add_stea := "Simulare".add_stea + 1; END_IF;
   "Simulare".paritate_stea := "Simulare".add_stea MOD 2.0;
   #_w2 := NOT "Ventilator".pornire_triunghi AND NOT "Avarii".avarie_ventilator AND "Ventilator".pornire_ventilator;
   "Variabile_HMI".stea_1 := #_w2 AND ("Simulare".paritate_stea = 0.0);
   "Variabile_HMI".stea_2 := #_w2 AND ("Simulare".paritate_stea = 1.0);
   IF "Simulare".resetare_cuptor THEN "Simulare".add_stea := 0; END_IF;
END_REGION

REGION Network 17: HMI ventilator triunghi
   RUNG wire#powerrail
      Contact( "Ventilator".pornire_triunghi )
      P_Contact(operand := "Clock_1Hz", bit := "Variabile_HMI".re_triunghi)
      Add(in1 := "Simulare".add_triunghi, in2 := 1.0, out => "Simulare".add_triunghi)
   END_RUNG
   RUNG wire#powerrail
      { S7_Templates := "SrcType := Int" } Mod(in1 := "Simulare".add_triunghi, in2 := 2.0, out => "Simulare".paritate_triunghi)
      I_Contact( "Ventilator".pornire_stea )
      I_Contact( "Avarii".avarie_ventilator )
      Contact( "Ventilator".pornire_ventilator )
      wire#w1
      { S7_Templates := "SrcType := Real" } EQ_Contact(in1 := "Simulare".paritate_triunghi, in2 := 0.0)
      Coil( "Variabile_HMI".triunghi_1 )
   END_RUNG
   RUNG wire#w1
      { S7_Templates := "SrcType := Real" } EQ_Contact(in1 := "Simulare".paritate_triunghi, in2 := 1.0)
      Coil( "Variabile_HMI".triunghi_2 )
   END_RUNG
   RUNG wire#powerrail
      Contact( "Simulare".resetare_cuptor )
      Move(in := 0, out1 => "Simulare".add_triunghi)
   END_RUNG
   // the same network as SCL:
   #_w1 := "Ventilator".pornire_triunghi AND "Clock_1Hz" AND NOT "Variabile_HMI".re_triunghi;   // rising edge of "Clock_1Hz"
   "Variabile_HMI".re_triunghi := "Clock_1Hz";
   IF #_w1 THEN "Simulare".add_triunghi := "Simulare".add_triunghi + 1.0; END_IF;
   "Simulare".paritate_triunghi := "Simulare".add_triunghi MOD 2.0;
   #_w2 := NOT "Ventilator".pornire_stea AND NOT "Avarii".avarie_ventilator AND "Ventilator".pornire_ventilator;
   "Variabile_HMI".triunghi_1 := #_w2 AND ("Simulare".paritate_triunghi = 0.0);
   "Variabile_HMI".triunghi_2 := #_w2 AND ("Simulare".paritate_triunghi = 1.0);
   IF "Simulare".resetare_cuptor THEN "Simulare".add_triunghi := 0; END_IF;
END_REGION
END_ORGANIZATION_BLOCK

(* ===== HMI "HMI_RT_1" =====
system functions are stored by id; their names below are inferred from use
connection "HMI_Connection_1": ETHERNET, SMART_S7_1500_OMS

HMI tags "Default tag table"
   "Tag_ScreenNumber" : UInt, internal
   "Simulare_temperatura_curenta" : Real = PLC Simulare.temperatura_curenta, 1 s
   "Alarme_alarm_gather" : Word = PLC Alarme.alarm_gather, 1 s
   "Usa_btn_usa_deschisa" : Bool = PLC Usa.btn_usa_deschisa, 1 s
   "Usa_usa_inchisa" : Bool = PLC Usa.usa_inchisa, 1 s
   "Usa_btn_usa_deschidere_urgenta" : Bool = PLC Usa.btn_usa_deschidere_urgenta, 1 s
   "Butoane_btn_pornire" : Bool = PLC Butoane.btn_pornire, 1 s
   "Simulare_resetare_cuptor" : Bool = PLC Simulare.resetare_cuptor, 1 s
   "Trapa_btn_trapa_deschisa" : Bool = PLC Trapa.btn_trapa_deschisa, 1 s
   "Trapa_btn_trapa_deschidere_urgenta" : Bool = PLC Trapa.btn_trapa_deschidere_urgenta, 1 s
   "Trapa_trapa_inchisa" : Bool = PLC Trapa.trapa_inchisa, 1 s
   "Ventilator_btn_pornire_urgenta" : Bool = PLC Ventilator.btn_pornire_urgenta, 1 s
   "Ventilator_pornire_ventilator" : Bool = PLC Ventilator.pornire_stea, 1 s
   "Arzator_arzator_pornit" : Bool = PLC Arzator.arzator_pornit, 1 s
   "Avarii_esd" : Bool = PLC Avarii.esd, 1 s
   "Avarii_esd_btn" : Bool = PLC Avarii.esd_btn, 1 s
   "Avarii_reset_esd_btn" : Bool = PLC Avarii.reset_esd_btn, 1 s
   "Avarii_avarie_usa" : Bool = PLC Avarii.avarie_usa, 1 s
   "Avarii_reset_avarie_generala_btn" : Bool = PLC Avarii.reset_avarie_generala_btn, 1 s
   "Avarii_avarie_generala" : Bool = PLC Avarii.avarie_generala, 1 s
   "Permisiuni_cuptor_terminat" : Bool = PLC Permisiuni.cuptor_terminat, 1 s
   "Simulare_timp_curent" : Time = PLC Simulare.timp_curent, 1 s
   "Simulare_timp_curent_hmi" : Time = PLC Simulare.timp_curent_hmi, 1 s
   "Alarme_alarm_vect{7}" : Bool = PLC Alarme.alarm_vect[7], 1 s
   "Simulare_temperatura_ceruta" : Real = PLC Simulare.temperatura_ceruta, 1 s
   "Simulare_timp_cuptor_ms" : Time = PLC Simulare.timp_cuptor_ms, 1 s
   "Avarii_avarie_trapa" : Bool = PLC Avarii.avarie_trapa, 1 s
   "Avarii_avarie_arzator" : Bool = PLC Avarii.avarie_arzator, 1 s
   "Avarii_avarie_ventilator" : Bool = PLC Avarii.avarie_ventilator, 1 s
   "Simulare_timp_cuptor" : Time = PLC Simulare.timp_cuptor, 1 s
   "Avarii_avarie_hmi" : Bool = PLC Avarii.avarie_hmi, 1 s
   "Ventilator_pornire_ventilator(1)" : Bool = PLC Ventilator.pornire_ventilator, 1 s
   "Variabile_HMI_stea_1" : Bool = PLC Variabile_HMI.stea_1, 1 s
   "Variabile_HMI_triunghi_1" : Bool = PLC Variabile_HMI.triunghi_1, 1 s
   "Variabile_HMI_stea_2" : Bool = PLC Variabile_HMI.stea_2, 1 s
   "Variabile_HMI_triunghi_2" : Bool = PLC Variabile_HMI.triunghi_2, 1 s
   "Ventilator_pornire_triunghi" : Bool = PLC Ventilator.pornire_triunghi, 1 s

discrete alarms
   1: 'ESD', class Errors, trigger "Alarme_alarm_gather" bit 0
   2: 'Avarie la usa', class Errors, trigger "Alarme_alarm_gather" bit 1
   3: 'Avarie la trapa de aerisire', class Errors, trigger "Alarme_alarm_gather" bit 2
   4: 'Avarie la arzator', class Errors, trigger "Alarme_alarm_gather" bit 3
   5: 'Avarie la ventilator', class Errors, trigger "Alarme_alarm_gather" bit 4
   6: 'Usa nu este inchisa, nu poate porni/continua', class Errors, trigger "Alarme_alarm_gather" bit 5
   7: 'Temperatura este prea mare, usa nu poate fi deschisa normal', class Errors, trigger "Alarme_alarm_gather" bit 6
   8: 'Produsul este gata sa fie scos din cuptor', class Errors, trigger "Alarme_alarm_gather" bit 7
   9: 'Produsul la 50%', class Errors, trigger "Alarme_alarm_gather" bit 8
   10: 'Produsul la 80%', class Errors, trigger "Alarme_alarm_gather" bit 9
   11: 'Produsul este gata, urmeaza racirea', class Errors, trigger "Alarme_alarm_gather" bit 10
   12: 'Timpul in cuptor nu a fost introdus', class Errors, trigger "Alarme_alarm_gather" bit 11
   13: 'Temperatura dorita nu a fost introdusa', class Errors, trigger "Alarme_alarm_gather" bit 12

recipe "Ciment": Temperatura <- "Simulare_temperatura_ceruta", Timp <- "Simulare_timp_cuptor_ms"

recipe "Moloz": Temperatura <- "Simulare_temperatura_ceruta", Timp <- "Simulare_timp_cuptor_ms"

Template "Template_1" 800x480
   Button "Exit" at 722,440 size 55x39; TextOff 'Exit'; PictureOff "ExitRuntime_KTP900_Basic_PN_TR"; PictureOn "ExitRuntime_KTP900_Basic_PN_TR"
      on Release: StopRuntime(0)
   Button "Alarms" at 622,440 size 55x39; TextOff 'Alarms'; PictureOff "AlarmDisplay_KTP900_Basic_PN_TR"; PictureOn "AlarmDisplay_KTP900_Basic_PN_TR"
      on Release: function_ef3f5d25("Alarm window_1", -1)
   Button "Start screen" at 522,440 size 55x39; TextOff 'Start screen'; PictureOff "NavigateHome_KTP900_Basic_PN_TR"; PictureOn "NavigateHome_KTP900_Basic_PN_TR"
      on Release: ActivateScreen("Simulare cuptor", 0)

screen "Simulare avarii" 800x480, template "Template_1"
   on GenerateScreen: SetTag("Tag_ScreenNumber", 1)
   TextField "Text field_1" at 18,455 size 60x20; Text 'Simulare'
   TextField "Text field_2" at 127,455 size 43x20; Text 'Avarii'
   TextField "Text field_3" at 230,455 size 42x20; Text 'Grafic'
   TextField "Text field_4" at 324,455 size 50x20; Text 'Retete'
   TextField "Text field_5" at 365,13 size 65x29; Text 'Avarii'
   Button "Button_14" at 50,393 size 96x32; TextOff 'Reset'
      on Click: SetBit("Avarii_reset_avarie_generala_btn")
   Circle "Circle_6" at 135,173 size 32x32
      Appearance <- "Avarii_avarie_usa"
   Button "Button_1" at 664,93 size 96x32; TextOff 'ESD'
      on Click: SetBit("Avarii_esd_btn")
   Button "Button_2" at 664,131 size 96x32; TextOff 'Reset'
      on Click: SetBit("Avarii_reset_esd_btn")
   Circle "Circle_1" at 693,41 size 38x38
      Appearance <- "Avarii_esd"
   TextField "Text field_16" at 423,455 size 44x20; Text 'Motor'
   TextField "Text field_6" at 69,128 size 59x20; Text 'Aparate'
   Button "Button_3" at 20,173 size 96x32; TextOff 'Usa'
      on Release: SetBit("Avarii_avarie_usa")
   Circle "Circle_2" at 135,228 size 32x32
      Appearance <- "Avarii_avarie_trapa"
   Button "Button_4" at 20,228 size 96x32; TextOff 'Trapa'
      on Release: SetBit("Avarii_avarie_trapa")
   Circle "Circle_3" at 135,281 size 32x32
      Appearance <- "Avarii_avarie_arzator"
   Button "Button_5" at 20,281 size 96x32; TextOff 'Aprinzator'
      on Release: SetBit("Avarii_avarie_arzator")
   Circle "Circle_4" at 135,336 size 32x32
      Appearance <- "Avarii_avarie_ventilator"
   Button "Button_6" at 20,336 size 96x32; TextOff 'Ventilator'
      on Release: SetBit("Avarii_avarie_ventilator")

screen "Simulare cuptor" 800x480
   TextField "Text field_1" at 18,455 size 60x20; Text 'Simulare'
   TextField "Text field_2" at 127,455 size 43x20; Text 'Avarii'
   TextField "Text field_3" at 230,455 size 42x20; Text 'Grafic'
   TextField "Text field_4" at 324,455 size 50x20; Text 'Retete'
   TextField "Text field_5" at 360,13 size 76x29; Text 'Cuptor'
   Button "Button_1" at 170,154 size 61x32; TextOff 'Deschis'
      on Release: SetBit("Usa_btn_usa_deschisa")
   Button "Button_2" at 170,188 size 62x32; TextOff 'Inchis'
      on Release: ResetBit("Usa_btn_usa_deschisa")
   TextField "Text field_6" at 185,131 size 28x20; Text 'Usa'
   Button "Button_3" at 700,305 size 39x32; TextOff 'On'
      on Release: SetBit("Usa_btn_usa_deschidere_urgenta")
   Button "Button_4" at 747,305 size 39x32; TextOff 'Off'
      on Release: ResetBit("Usa_btn_usa_deschidere_urgenta")
   TextField "Text field_7" at 633,313 size 28x20; Text 'Usa'
   Button "Button_5" at 19,212 size 58x32; TextOff 'Pornire'
      on Release: SetBit("Butoane_btn_pornire")
   Button "Button_6" at 92,212 size 64x32; TextOff 'Restart'
      on Release: SetBit("Simulare_resetare_cuptor")
   Button "Button_9" at 700,363 size 39x32; TextOff 'On'
      on Release: SetBit("Trapa_btn_trapa_deschidere_urgenta")
   Button "Button_10" at 747,362 size 39x32; TextOff 'Off'
      on Release: ResetBit("Trapa_btn_trapa_deschidere_urgenta")
   TextField "Text field_9" at 628,369 size 42x20; Text 'Trapa'
   Button "Button_7" at 700,423 size 39x32; TextOff 'On'
      on Release: SetBit("Ventilator_btn_pornire_urgenta")
   Button "Button_8" at 747,423 size 39x32; TextOff 'Off'
      on Release: ResetBit("Ventilator_btn_pornire_urgenta")
   TextField "Text field_8" at 617,429 size 70x20; Text 'Ventilator'
   Button "Button_11" at 664,93 size 96x32; TextOff 'ESD'
      on Click: SetBit("Avarii_esd_btn")
   Button "Button_12" at 664,131 size 96x32; TextOff 'Reset'
      on Click: SetBit("Avarii_reset_esd_btn")
   Circle "Circle_5" at 693,41 size 38x38
      Appearance <- "Avarii_esd"
   Rectangle "Rectangle_4" at 243,140 size 44x158
      Appearance <- "Usa_usa_inchisa"
   Rectangle "Rectangle_5" at 510,125 size 19x194
      Appearance <- "Ventilator_pornire_ventilator(1)"
   Rectangle "Rectangle_6" at 339,95 size 159x14
      Appearance <- "Trapa_trapa_inchisa"
   Rectangle "Rectangle_7" at 379,327 size 37x19
      Appearance <- "Arzator_arzator_pornit"
   TextField "Text field_10" at 396,73 size 42x20; Text 'Trapa'
   TextField "Text field_11" at 529,154 size 70x20; Text 'Ventilator'
   TextField "Text field_12" at 369,346 size 56x20; Text 'Arzator'
   TextField "Text field_13" at 23,51 size 275x20; Text 'Produsul este gata sa fie scos din cuptor!'
      Visibility <- "Alarme_alarm_vect{7}"
   IOField "I/O field_1" at 348,163 size 96x32; FormatPattern 99.99; Unit °C
      ProcessValue <- "Simulare_temperatura_curenta"
   IOField "I/O field_2" at 349,244 size 96x32; FormatPattern 999; Unit s
      ProcessValue <- "Simulare_timp_curent_hmi"
   TextField "Text field_14" at 328,140 size 144x20; Text 'Temperatura curenta'
   TextField "Text field_15" at 350,222 size 92x20; Text 'Timpul curent'
   TextField "Text field_16" at 423,455 size 44x20; Text 'Motor'
   TextField "Text field_17" at 672,260 size 71x23; Text 'Urgente'
   TextField "Text field_18" at 67,263 size 53x23; Text 'Valori'
   IOField "I/O field_3" at 82,319 size 96x32; FormatPattern 999.99; Unit °C
      ProcessValue <- "Simulare_temperatura_ceruta"
   IOField "I/O field_4" at 82,378 size 96x32; FormatPattern 999; Unit s
      ProcessValue <- "Simulare_timp_cuptor_ms"
   TextField "Text field_19" at 19,322 size 43x20; Text 'Temp.'
   TextField "Text field_20" at 22,383 size 34x20; Text 'Timp'
   Circle "Circle_1" at 63,141 size 48x48
      Appearance <- "Avarii_avarie_generala"
   TextField "Text field_21" at 63,116 size 48x20; Text 'Avarie'
   TextField "Text field_22" at 23,64 size 274x20; Text 'Avarie, scoateti produsul daca este cazul'
      Visibility <- "Avarii_avarie_hmi"

screen "Grafic" 800x480
   TrendView "Trend view_1" at 0,64 size 800x355
   TextField "Text field_1" at 18,455 size 60x20; Text 'Simulare'
   TextField "Text field_2" at 127,455 size 43x20; Text 'Avarii'
   TextField "Text field_3" at 230,455 size 42x20; Text 'Grafic'
   TextField "Text field_4" at 324,455 size 50x20; Text 'Retete'
   TextField "Text field_5" at 295,13 size 215x29; Text 'Temperatura cuptor'
   TextField "Text field_16" at 423,455 size 44x20; Text 'Motor'

screen "Retete" 800x480
   TextField "Text field_1" at 18,455 size 60x20; Text 'Simulare'
   TextField "Text field_2" at 127,455 size 43x20; Text 'Avarii'
   TextField "Text field_3" at 230,455 size 42x20; Text 'Grafic'
   TextField "Text field_4" at 324,455 size 50x20; Text 'Retete'
   TextField "Text field_5" at 364,13 size 74x29; Text 'Retete'
   Button "Button_11" at 664,93 size 96x32; TextOff 'ESD'
      on Click: SetBit("Avarii_esd_btn")
   Button "Button_12" at 664,131 size 96x32; TextOff 'Reset'
      on Click: SetBit("Avarii_reset_esd_btn")
   Circle "Circle_5" at 693,41 size 38x38
      Appearance <- "Avarii_esd"
   TextField "Text field_16" at 423,455 size 44x20; Text 'Motor'
   RecipeView "Recipe view_1" at 43,68 size 590x356

screen "Motor_ventilator" 800x480
   TextField "Text field_1" at 18,455 size 60x20; Text 'Simulare'
   TextField "Text field_2" at 127,455 size 43x20; Text 'Avarii'
   TextField "Text field_3" at 230,455 size 42x20; Text 'Grafic'
   TextField "Text field_4" at 324,455 size 50x20; Text 'Retete'
   Button "Button_11" at 664,93 size 96x32; TextOff 'ESD'
      on Click: SetBit("Avarii_esd_btn")
   Button "Button_12" at 664,131 size 96x32; TextOff 'Reset'
      on Click: SetBit("Avarii_reset_esd_btn")
   Circle "Circle_5" at 693,41 size 38x38
      Appearance <- "Avarii_esd"
   TextField "Text field_16" at 423,455 size 44x20; Text 'Motor'
   GraphicView "Graphic view_1" at 104,79 size 306x295; Picture "Graphic_1"
      Visibility <- "Ventilator_pornire_ventilator(1)"
   GraphicView "Graphic view_2" at 105,79 size 306x296; Picture "Graphic_2"
      Visibility <- "Variabile_HMI_stea_1"
   GraphicView "Graphic view_7" at 105,79 size 306x296; Picture "Graphic_8"
      Visibility <- "Variabile_HMI_stea_2"
   GraphicView "Graphic view_6" at 105,78 size 306x296; Picture "Graphic_3"
      Visibility <- "Variabile_HMI_triunghi_2"
   GraphicView "Graphic view_8" at 105,78 size 306x296; Picture "Graphic_9"
      Visibility <- "Avarii_avarie_ventilator"
   TextField "Text field_5" at 655,251 size 37x20; Text 'Oprit'
   TextField "Text field_6" at 651,289 size 48x20; Text 'Avarie'
   TextField "Text field_7" at 657,330 size 35x20; Text 'Stea'
   TextField "Text field_8" at 645,370 size 56x20; Text 'Triunghi'
   Button "Button_7" at 700,423 size 39x32; TextOff 'On'
      on Release: SetBit("Ventilator_btn_pornire_urgenta")
   Button "Button_8" at 747,423 size 39x32; TextOff 'Off'
      on Release: ResetBit("Ventilator_btn_pornire_urgenta")
   TextField "Text field_9" at 617,429 size 70x20; Text 'Ventilator'
   Button "Button_14" at 549,131 size 96x32; TextOff 'Reset'
      on Click: SetBit("Avarii_reset_avarie_generala_btn")
   Button "Button_6" at 549,93 size 96x32; TextOff 'Ventilator'
      on Release: SetBit("Avarii_avarie_ventilator")
   GraphicView "Graphic view_4" at 104,78 size 308x297; Picture "Graphic_10"
      Visibility <- "Variabile_HMI_triunghi_1"
   Circle "Circle_1" at 721,245 size 32x32
      Appearance <- "Ventilator_pornire_ventilator(1)"
   Circle "Circle_2" at 721,285 size 32x32
      Appearance <- "Avarii_avarie_ventilator"
   Circle "Circle_3" at 721,325 size 32x32
      Appearance <- "Ventilator_pornire_ventilator"
   Circle "Circle_6" at 721,365 size 32x32
      Appearance <- "Ventilator_pornire_triunghi"
   TextField "Text field_10" at 569,52 size 58x23; Text 'Avarie'
*)